// Mitsubishi GX Works2 project: AutomationProject (1)   PLC: FX3G

// global labels: Global1
VAR_GLOBAL
  StartWorkingDay AT X007 : BOOL;
  InputRaspberry AT D1101 : REAL;
  StockRaspberry AT D1109 : REAL;
  InputLemon AT D1103 : REAL;
  StockLemon AT D1111 : REAL;
  InputStabelizer AT D1105 : REAL;
  InputStabilizer AT D1105 : REAL;
  StockStabilizer AT D1113 : REAL;
  InputGummyBears AT D1107 : REAL;
  StockGummyBears AT D1115 : REAL;
END_VAR
VAR_GLOBAL CONSTANT
  ResetWord : INT := K0;
END_VAR
VAR_GLOBAL
  AnalogOutPut AT D8282 : INT;
  PacksContainer AT D1129 : REAL;
  Reset AT X010 : BOOL;
  ResetBtn AT X010 : BOOL;
  EmergencyBtn AT X005 : BOOL;
  M_20 AT M20 : BOOL;
END_VAR
VAR_GLOBAL CONSTANT
  ResetVal : REAL;
END_VAR
VAR_GLOBAL
  MaterialCheck AT X001 : BOOL;
  AnalogInput AT D8280 : INT;
  FloatInput AT D1119 : REAL;
  FlaotInput AT D119 : REAL;
  M_25 AT M25 : BOOL;
END_VAR
VAR_GLOBAL CONSTANT
  Const5 : REAL := E5.0;
END_VAR
VAR_GLOBAL
  FinishPacking AT M50 : BOOL;
  EmergencyBth AT X005 : BOOL;
  RegularChoice AT M26 : BOOL;
  PinukChoice AT M27 : BOOL;
END_VAR
VAR_GLOBAL CONSTANT
  MinRegRasp : REAL := E280.0;
END_VAR
VAR_GLOBAL
  M_31 AT M31 : BOOL;
END_VAR
VAR_GLOBAL CONSTANT
  MinRegLemon : REAL := E455.0;
END_VAR
VAR_GLOBAL
  M_32 AT M32 : BOOL;
END_VAR
VAR_GLOBAL CONSTANT
  MinRegStab : REAL := E105.0;
END_VAR
VAR_GLOBAL
  M_33 AT M33 : BOOL;
END_VAR
VAR_GLOBAL CONSTANT
  MinRegGummy : REAL := E14.0;
END_VAR
VAR_GLOBAL
  M_34 AT M34 : BOOL;
END_VAR
VAR_GLOBAL CONSTANT
  MinPinRasp : REAL := E385.0;
END_VAR
VAR_GLOBAL
  M_41 AT M41 : BOOL;
END_VAR
VAR_GLOBAL CONSTANT
  MinPinLemon : REAL := E665.0;
END_VAR
VAR_GLOBAL
  M_42 AT M42 : BOOL;
END_VAR
VAR_GLOBAL CONSTANT
  MinPinStab : REAL := E210.0;
END_VAR
VAR_GLOBAL
  M_43 AT M43 : BOOL;
END_VAR
VAR_GLOBAL CONSTANT
  MinPinGummy : REAL := E35.0;
END_VAR
VAR_GLOBAL
  M_44 AT M44 : BOOL;
  M_30 AT M30 : BOOL;
  M_40 AT M40 : BOOL;
  M_100 AT M100 : BOOL;
  WorkingDay AT Y007 : BOOL;
  ValidForRegular AT M30 : BOOL;
  ValidForPinuk AT M40 : BOOL;
  NoValidMaterials AT M100 : BOOL;
  FlavorTimer AT TC1 : BOOL;
END_VAR
VAR_GLOBAL CONSTANT
  Flavour5Sec : INT := K50;
END_VAR
VAR_GLOBAL
  FinishFlavour AT TS1 : BOOL;
  FlavourMaker AT Y000 : BOOL;
  M_26 AT M26 : BOOL;
  M_27 AT M27 : BOOL;
  RaspIceCreamCont AT D1121 : REAL;
END_VAR
VAR_GLOBAL CONSTANT
  RegulaRasprCont : REAL := E350.0;
END_VAR
VAR_GLOBAL
  LemonIceCreamCont AT D1123 : REAL;
END_VAR
VAR_GLOBAL CONSTANT
  RegulaLemonCont : REAL := E490.0;
  PinukRasprCont : REAL := E560.0;
  PinukLemonCont : REAL := E700.0;
END_VAR
VAR_GLOBAL
  M_60 AT M60 : BOOL;
  FinishFlavourProcess AT M61 : BOOL;
  M_66 AT M66 : BOOL;
  M_61 AT M61 : BOOL;
  ColdRaspCont AT D1125 : REAL;
  ColdLemoCont AT D1127 : REAL;
  FinishMoveToCool AT M62 : BOOL;
  ColdBtn AT X002 : BOOL;
  ColdLemonCont AT D1127 : REAL;
  ColdTimer AT TC2 : BOOL;
END_VAR
VAR_GLOBAL CONSTANT
  Cold8Sec : INT := K80;
END_VAR
VAR_GLOBAL
  FinishCold AT TS2 : BOOL;
  TempBtn AT X003 : BOOL;
  ColdMaker AT Y002 : BOOL;
  FinishColdProcess AT M63 : BOOL;
  MixingCont AT D1131 : REAL;
  M_64 AT M64 : BOOL;
  M_63 AT M63 : BOOL;
  LightRegTimer AT TC3 : BOOL;
END_VAR
VAR_GLOBAL CONSTANT
  MixReg : INT := K30;
END_VAR
VAR_GLOBAL
  FinishLightReg AT TS3 : BOOL;
  M_26_1 AT M70 : BOOL;
  M_27_1 AT M71 : BOOL;
END_VAR
VAR_GLOBAL CONSTANT
  MixPinuk : INT := K50;
END_VAR
VAR_GLOBAL
  Timer_1 AT K10 : INT;
  M_81 AT M81 : BOOL;
  LightPinTimer AT TC4 : BOOL;
  FinishLighPin AT TS4 : BOOL;
  Y_5 AT Y005 : BOOL;
  TC_6 AT TC6 : BOOL;
  TS_6 AT TS6 : BOOL;
  Y_6 AT Y006 : BOOL;
  TC_8 AT TC8 : BOOL;
  TS_8 AT TS8 : BOOL;
  TC_9 AT TC9 : BOOL;
  TS_9 AT TS9 : BOOL;
  M_82 AT M82 : BOOL;
  TC_10 AT TC10 : BOOL;
  TS_10 AT TS10 : BOOL;
  FinishLightPin AT TS4 : BOOL;
END_VAR
VAR_GLOBAL CONSTANT
  Const1 : REAL := E1.0;
  Const40 : REAL := E40.0;
END_VAR
VAR_GLOBAL
  Packages AT D1133 : REAL;
  M_75 AT M75 : BOOL;
  M_76 AT M76 : BOOL;
  TC_11 AT TC11 : BOOL;
  TS_11 AT TS11 : BOOL;
  TC_12 AT TC12 : BOOL;
  TS_12 AT TS12 : BOOL;
  M_88 AT M88 : BOOL;
  TS_4 AT TS4 : BOOL;
  TS_3 AT TS3 : BOOL;
END_VAR

// task Task_01 (event TRUE, interval 0, priority 31): POU_01

PROGRAM POU_01
VAR CONSTANT
  DIV400 : REAL := E400;
END_VAR
(* structured ladder/FBD written out as ST: instructions are called as NAME(EN, inputs, outputs); _pN, _eN, _tN stand for wires *)
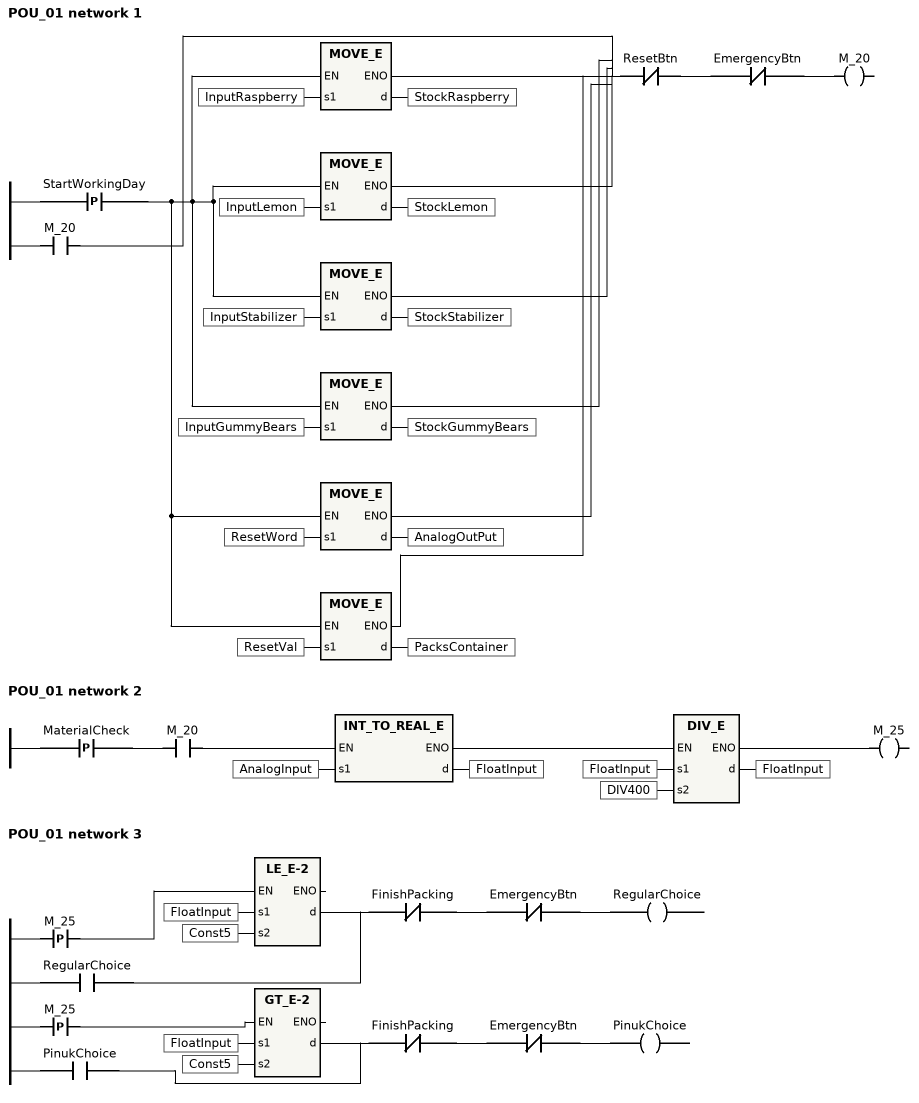
(* network 1 *)
_p1 := LDP(TRUE, StartWorkingDay);
_e2 := MOVE_E(_p1, InputRaspberry, StockRaspberry);
_e3 := MOVE_E(_p1, InputLemon, StockLemon);
_e4 := MOVE_E(_p1, InputStabilizer, StockStabilizer);
_e5 := MOVE_E(_p1, InputGummyBears, StockGummyBears);
_e6 := MOVE_E(_p1, ResetWord, AnalogOutPut);
_e7 := MOVE_E(_p1, ResetVal, PacksContainer);
M_20 := ((_e2 OR _e3 OR _e4 OR _e5 OR _e6 OR _e7 OR M_20) AND NOT ResetBtn) AND NOT EmergencyBtn;
(* network 2 *)
_e1 := INT_TO_REAL_E(LDP(TRUE, MaterialCheck) AND M_20, AnalogInput, FloatInput);
_e2 := DIV_E(_e1, FloatInput, DIV400, FloatInput);
M_25 := _e2;
(* network 3 *)
LE_E(LDP(TRUE, M_25), FloatInput, Const5, _t1);
RegularChoice := ((_t1 OR RegularChoice) AND NOT FinishPacking) AND NOT EmergencyBtn;
GT_E(LDP(TRUE, M_25), FloatInput, Const5, _t2);
PinukChoice := ((_t2 OR PinukChoice) AND NOT FinishPacking) AND NOT EmergencyBtn;
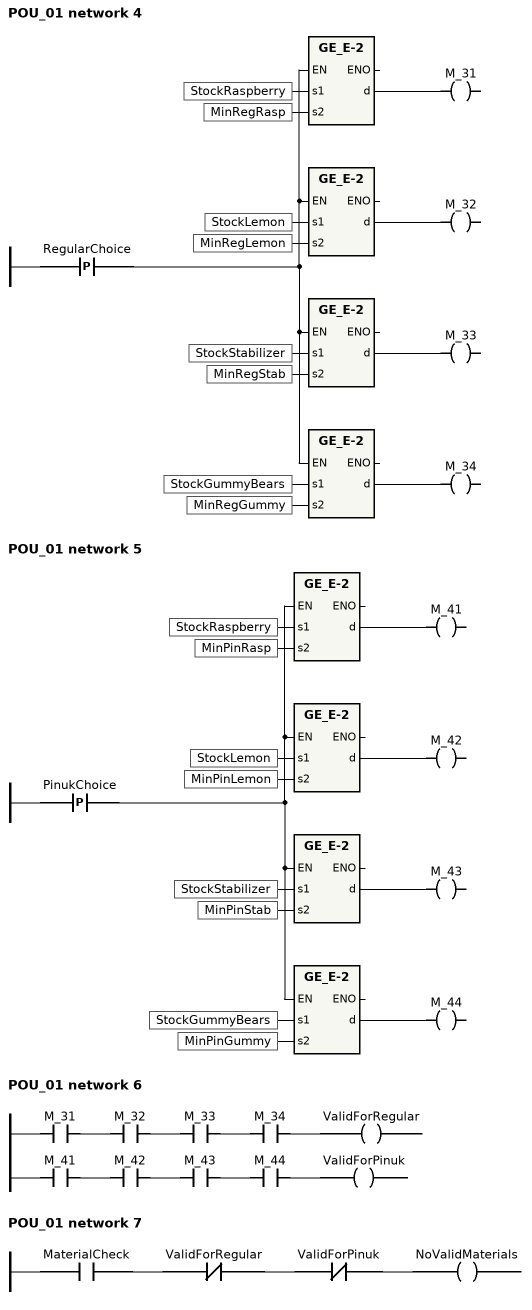
(* network 4 *)
_p1 := LDP(TRUE, RegularChoice);
GE_E(_p1, StockRaspberry, MinRegRasp, _t2);
M_31 := _t2;
GE_E(_p1, StockLemon, MinRegLemon, _t3);
M_32 := _t3;
GE_E(_p1, StockStabilizer, MinRegStab, _t4);
M_33 := _t4;
GE_E(_p1, StockGummyBears, MinRegGummy, _t5);
M_34 := _t5;
(* network 5 *)
_p1 := LDP(TRUE, PinukChoice);
GE_E(_p1, StockRaspberry, MinPinRasp, _t2);
M_41 := _t2;
GE_E(_p1, StockLemon, MinPinLemon, _t3);
M_42 := _t3;
GE_E(_p1, StockStabilizer, MinPinStab, _t4);
M_43 := _t4;
GE_E(_p1, StockGummyBears, MinPinGummy, _t5);
M_44 := _t5;
(* network 6 *)
ValidForRegular := M_31 AND M_32 AND M_33 AND M_34;
ValidForPinuk := M_41 AND M_42 AND M_43 AND M_44;
(* network 7 *)
NoValidMaterials := MaterialCheck AND NOT ValidForRegular AND NOT ValidForPinuk;
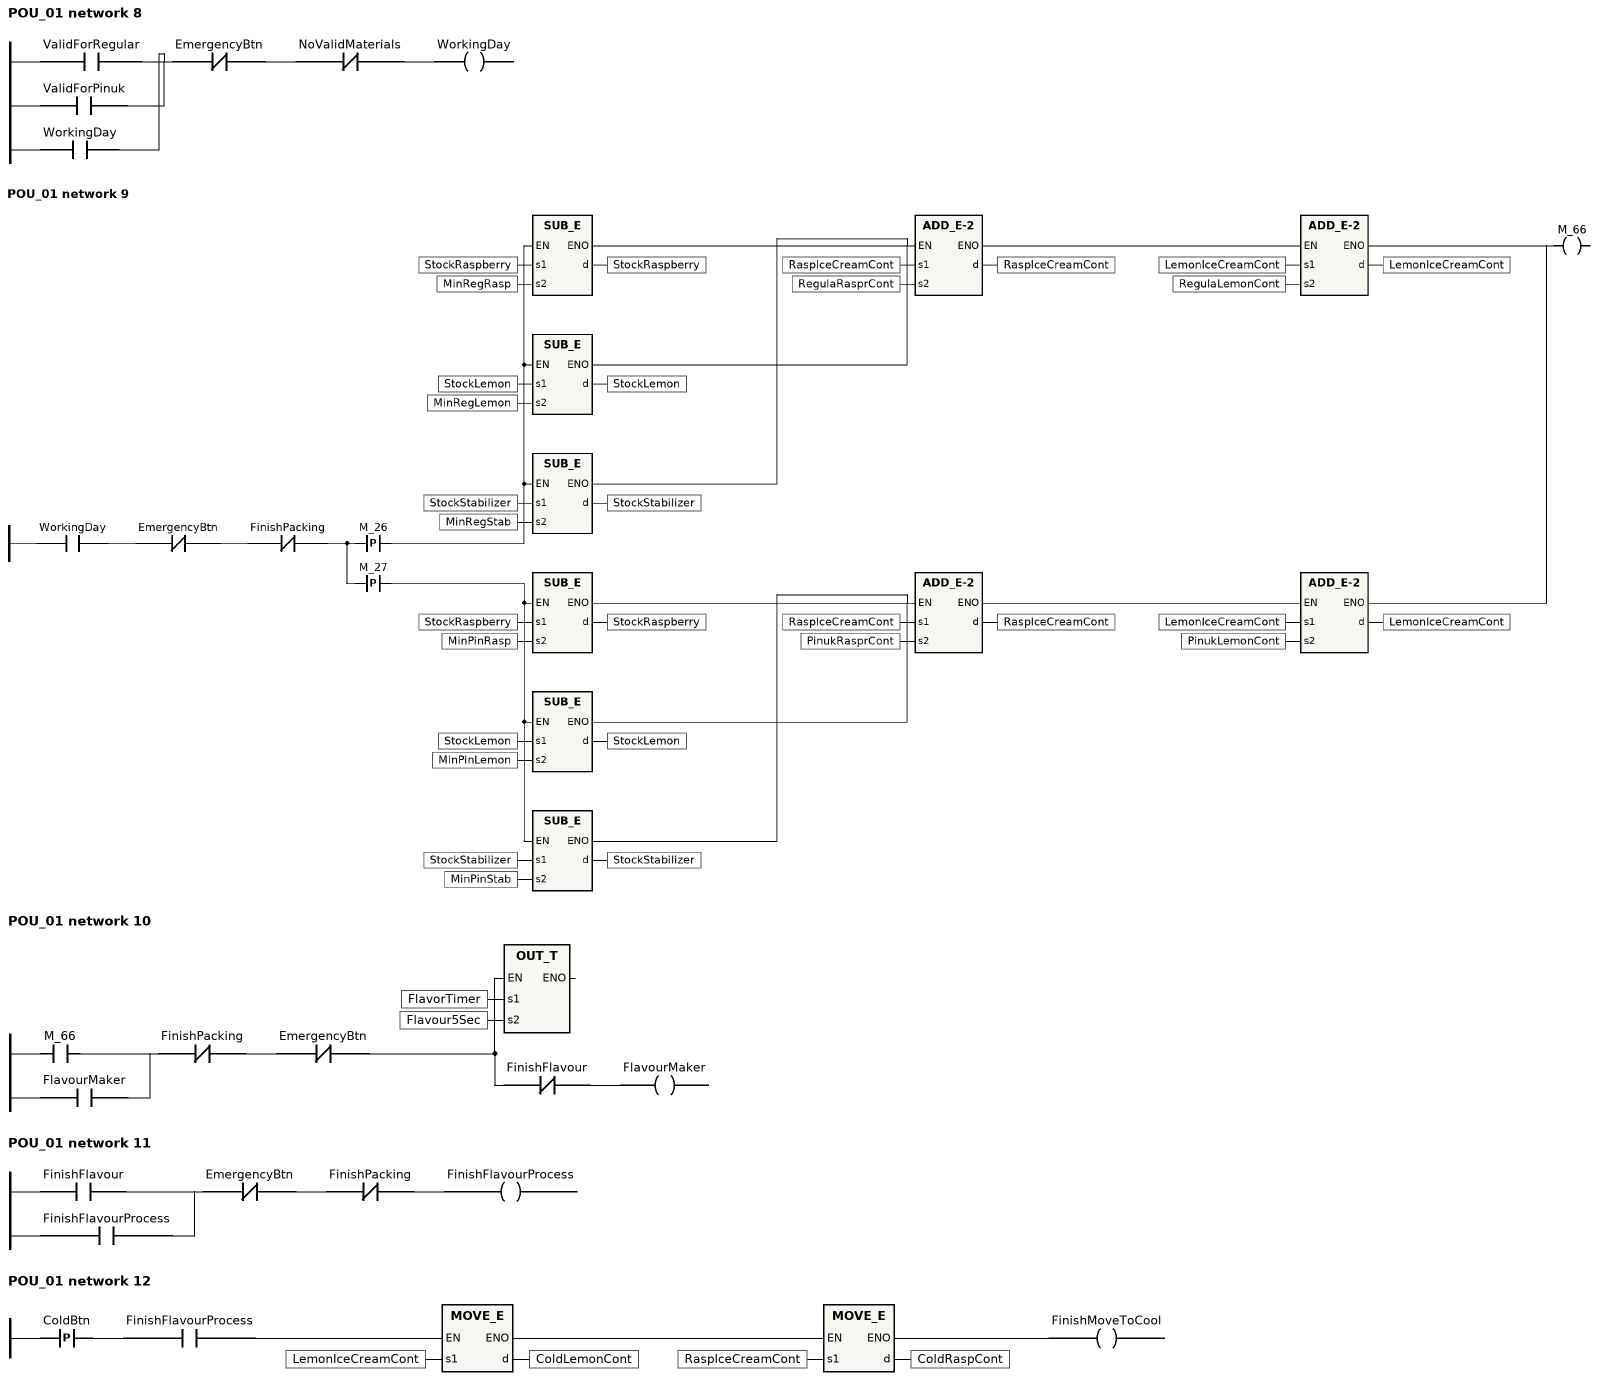
(* network 8 *)
WorkingDay := ((ValidForRegular OR ValidForPinuk OR WorkingDay) AND NOT EmergencyBtn) AND NOT NoValidMaterials;
(* network 9 *)
_p1 := WorkingDay AND NOT EmergencyBtn AND NOT FinishPacking;
_p2 := _p1 AND LDP(TRUE, M_26);
_e3 := SUB_E(_p2, StockRaspberry, MinRegRasp, StockRaspberry);
_e4 := SUB_E(_p2, StockLemon, MinRegLemon, StockLemon);
_e5 := SUB_E(_p2, StockStabilizer, MinRegStab, StockStabilizer);
_e6 := ADD_E(_e3 OR _e4 OR _e5, RaspIceCreamCont, RegulaRasprCont, RaspIceCreamCont);
_e7 := ADD_E(_e6, LemonIceCreamCont, RegulaLemonCont, LemonIceCreamCont);
_p8 := _p1 AND LDP(TRUE, M_27);
_e9 := SUB_E(_p8, StockRaspberry, MinPinRasp, StockRaspberry);
_e10 := SUB_E(_p8, StockLemon, MinPinLemon, StockLemon);
_e11 := SUB_E(_p8, StockStabilizer, MinPinStab, StockStabilizer);
_e12 := ADD_E(_e9 OR _e10 OR _e11, RaspIceCreamCont, PinukRasprCont, RaspIceCreamCont);
_e13 := ADD_E(_e12, LemonIceCreamCont, PinukLemonCont, LemonIceCreamCont);
M_66 := _e7 OR _e13;
(* network 10 *)
_p1 := ((M_66 OR FlavourMaker) AND NOT FinishPacking) AND NOT EmergencyBtn;
OUT_T(_p1, FlavorTimer, Flavour5Sec);
FlavourMaker := _p1 AND NOT FinishFlavour;
(* network 11 *)
FinishFlavourProcess := ((FinishFlavour OR FinishFlavourProcess) AND NOT EmergencyBtn) AND NOT FinishPacking;
(* network 12 *)
_e1 := MOVE_E(LDP(TRUE, ColdBtn) AND FinishFlavourProcess, LemonIceCreamCont, ColdLemonCont);
_e2 := MOVE_E(_e1, RaspIceCreamCont, ColdRaspCont);
FinishMoveToCool := _e2;
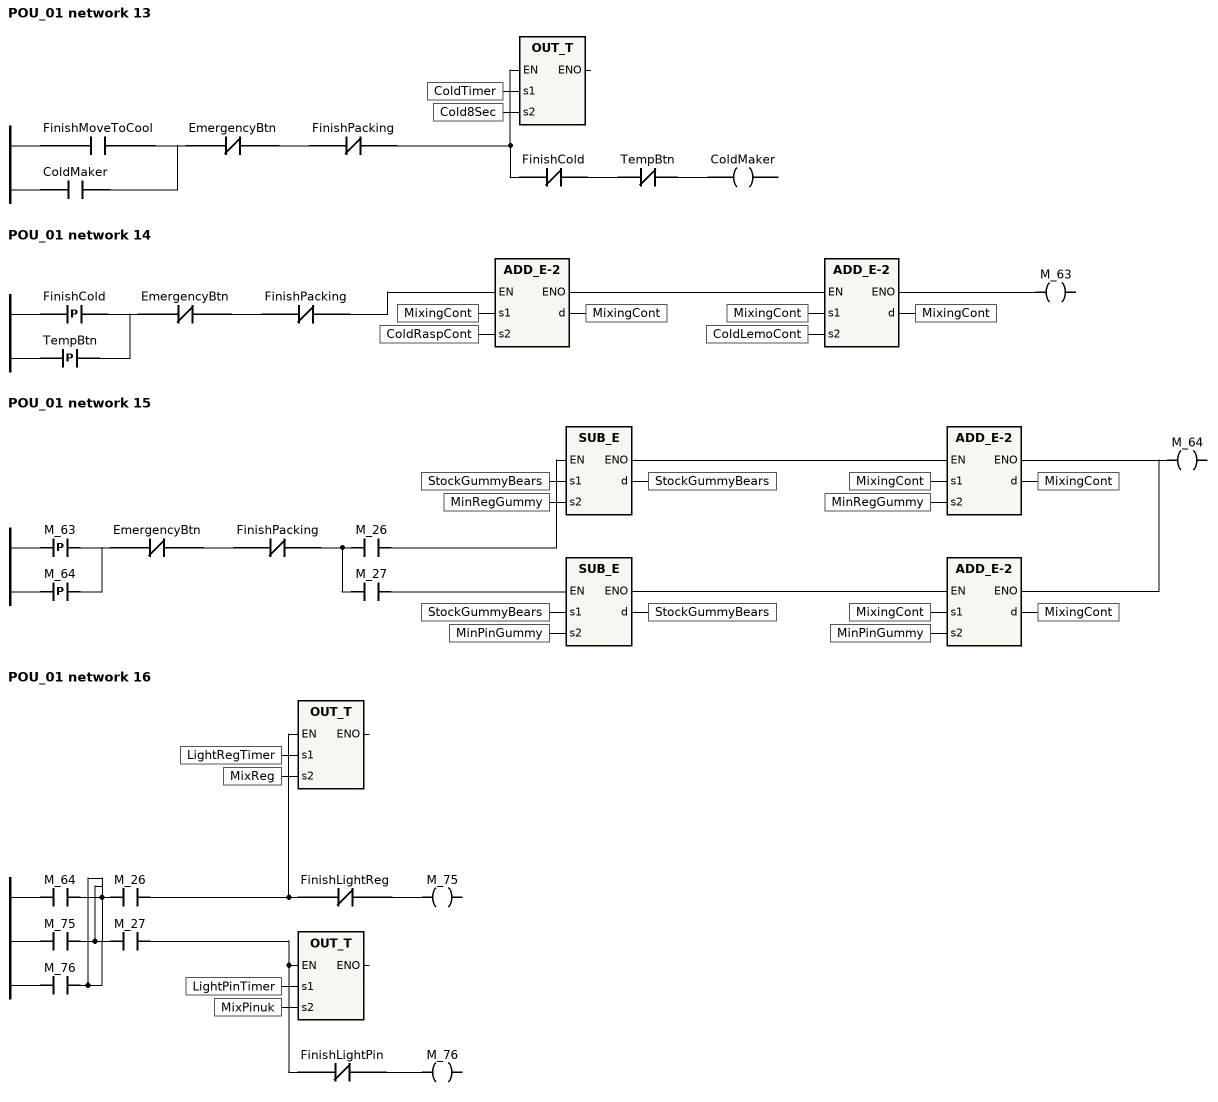
(* network 13 *)
_p1 := ((FinishMoveToCool OR ColdMaker) AND NOT EmergencyBtn) AND NOT FinishPacking;
OUT_T(_p1, ColdTimer, Cold8Sec);
ColdMaker := _p1 AND NOT FinishCold AND NOT TempBtn;
(* network 14 *)
_e1 := ADD_E(((LDP(TRUE, FinishCold) OR LDP(TRUE, TempBtn)) AND NOT EmergencyBtn) AND NOT FinishPacking, MixingCont, ColdRaspCont, MixingCont);
_e2 := ADD_E(_e1, MixingCont, ColdLemoCont, MixingCont);
M_63 := _e2;
(* network 15 *)
_p1 := ((LDP(TRUE, M_63) OR LDP(TRUE, M_64)) AND NOT EmergencyBtn) AND NOT FinishPacking;
_e2 := SUB_E(_p1 AND M_26, StockGummyBears, MinRegGummy, StockGummyBears);
_e3 := ADD_E(_e2, MixingCont, MinRegGummy, MixingCont);
_e4 := SUB_E(_p1 AND M_27, StockGummyBears, MinPinGummy, StockGummyBears);
_e5 := ADD_E(_e4, MixingCont, MinPinGummy, MixingCont);
M_64 := _e3 OR _e5;
(* network 16 *)
_p1 := M_64 OR M_75 OR M_76;
_p2 := _p1 AND M_26;
OUT_T(_p2, LightRegTimer, MixReg);
M_75 := _p2 AND NOT FinishLightReg;
_p3 := _p1 AND M_27;
OUT_T(_p3, LightPinTimer, MixPinuk);
M_76 := _p3 AND NOT FinishLightPin;
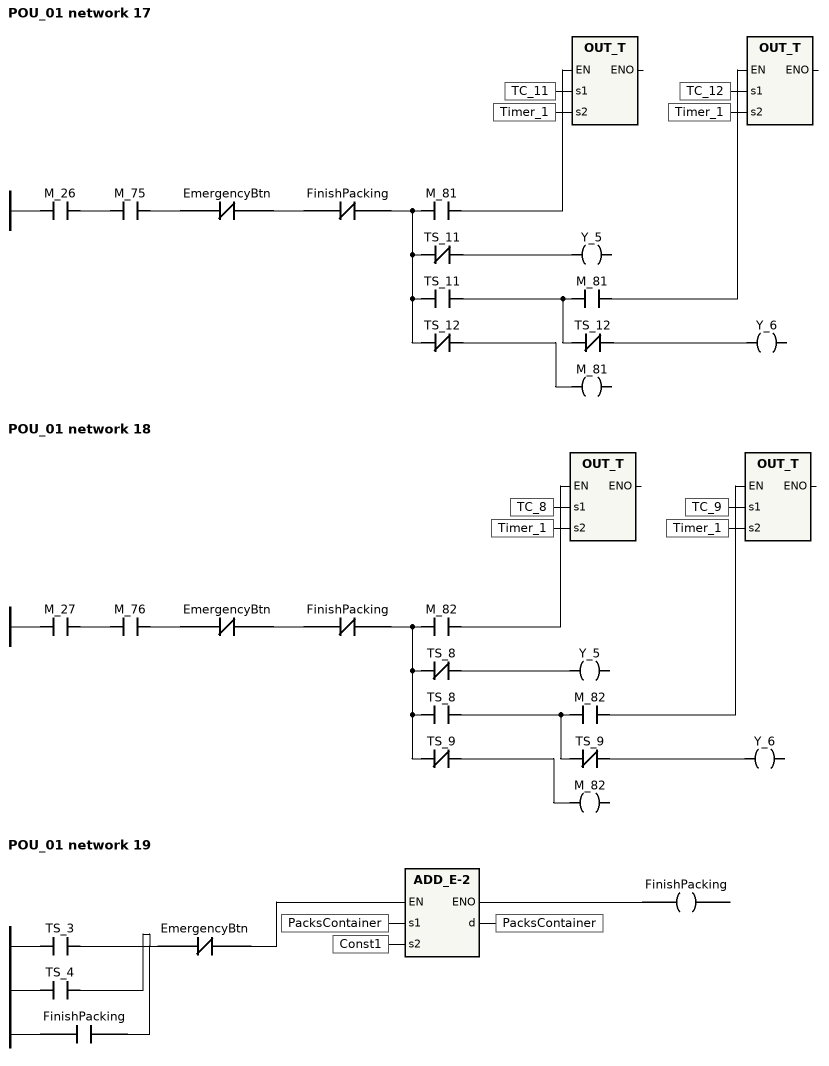
(* network 17 *)
_p1 := M_26 AND M_75 AND NOT EmergencyBtn AND NOT FinishPacking;
OUT_T(_p1 AND M_81, TC_11, Timer_1);
Y_5 := _p1 AND NOT TS_11;
_p2 := _p1 AND TS_11;
OUT_T(_p2 AND M_81, TC_12, Timer_1);
Y_6 := _p2 AND NOT TS_12;
M_81 := _p1 AND NOT TS_12;
(* network 18 *)
_p1 := M_27 AND M_76 AND NOT EmergencyBtn AND NOT FinishPacking;
OUT_T(_p1 AND M_82, TC_8, Timer_1);
Y_5 := _p1 AND NOT TS_8;
_p2 := _p1 AND TS_8;
OUT_T(_p2 AND M_82, TC_9, Timer_1);
Y_6 := _p2 AND NOT TS_9;
M_82 := _p1 AND NOT TS_9;
(* network 19 *)
_e1 := ADD_E((TS_3 OR TS_4 OR FinishPacking) AND NOT EmergencyBtn, PacksContainer, Const1, PacksContainer);
FinishPacking := _e1;
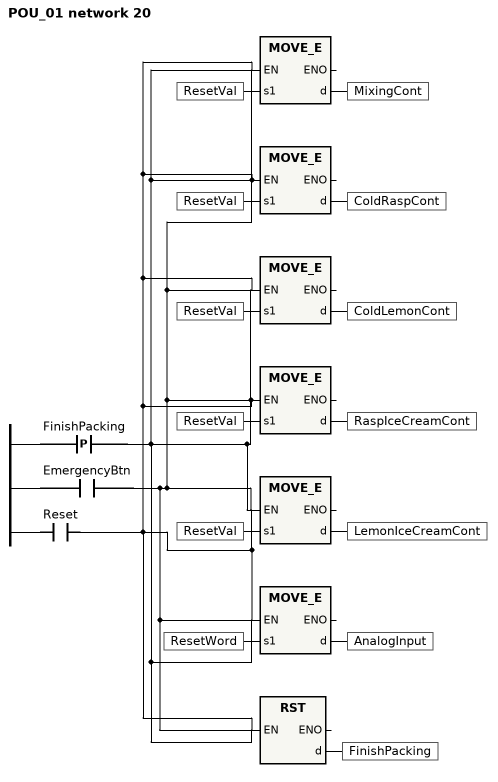
(* network 20 *)
_p1 := LDP(TRUE, FinishPacking) OR EmergencyBtn OR Reset;
MOVE_E(_p1, ResetVal, MixingCont);
MOVE_E(_p1, ResetVal, ColdRaspCont);
MOVE_E(_p1, ResetVal, ColdLemonCont);
MOVE_E(_p1, ResetVal, RaspIceCreamCont);
MOVE_E(_p1, ResetVal, LemonIceCreamCont);
MOVE_E(_p1, ResetWord, AnalogInput);
RST(_p1, FinishPacking);
END_PROGRAM
